// TIA Portal V17 export
// export: Created 2024-06-16T17:47:23.70489Z, ExportSetting WithDefaults, DisplayName Totally Integrated Automation Portal, DisplayVersion V17, DisplayName TIA Portal Openness, DisplayVersion V17, DisplayName TIA Portal Version Control Interface, DisplayVersion V17, DisplayName STEP 7 Professional, DisplayVersion V17, DisplayName STEP 7 Safety, DisplayVersion V17, DisplayName WinCC Professional, DisplayVersion V17
DATA_BLOCK "S00_Mode"   // DB1010
VERSION : 0.1
// stored: AutoNumber false, DBAccessibleFromOPCUA true, DBAccessibleFromWebserver true, InstanceOfName S00_Mode_FB, InstanceOfType FB
"S00_Mode_FB"
   // VAR_OUTPUT
   //    "Step" : Int;
   // END_VAR
   // VAR
   //    Step_100 : Int;
   //    Auto : Bool;
   //    Manu : Bool;
   //    PaP : Bool;
   // END_VAR
BEGIN
END_DATA_BLOCK
